// SIMATIC S7-200 project (STEP 7-Micro/WIN), CPU 224 CN REL 02.01

ORGANIZATION_BLOCK 补水控制:OB1
TITLE=我为200方给水净化工程设计了一个自动化控制系统，适用于自来水厂等场景。通过操作员按下启动按钮启动补水流程，并在未按下停止按钮时运行，确保供水质量和稳定性。
// 系统中涉及的物理设备包括补水泵1、补水泵2、进水阀、出水阀、余氯调节泵、水箱、启动按钮、停止按钮、水位传感器和阀门限位开关。
// Network 1开始，当启动按钮按下且停止按钮未按下时，若水位低传感器未触发，补水泵1启动，需通过定时器延时60个单位停止。
// Network 2中，补水泵2在水位高传感器未触发且标志位为真时启动，同样使用定时器延时停止。
// Network 3和Network 7通过定时器实现补水泵延时600个单位停止，确保水位恢复后泵不会立即停机。
// Network 16调用子程序，其中阀门控制根据阀门开限位和关限位控制进水阀和出水阀，要求动作在限位信号正确时执行。同时，进水阀和出水阀互锁防止同时开启。
// 当进水控制信号为真且阀门切换标志为假时，打开进水阀，以向水箱供水。
// 当出水控制信号为真时，打开出水阀，以排出水箱中的水。
// 余氯控制根据余氯浓度调节余氯调节泵，浓度低于7时启动，高于15时停止。
// 参数显示通过定时器每20个单位更新水质参数，并在触摸屏显示。
// PID控制根据补水泵状态调整模拟量输出，实现水流稳定。
// 
BEGIN
Network 1 // 网络标题
// 网络注释
LD     I0.0
AN     I0.1
AN     I0.2
AN     I2.1
AN     M0.0
LPS
A      T120
=      Q0.0
LPP
TON    T120, +60
Network 2
LD     I0.0
AN     I0.1
AN     I0.3
AN     I2.1
A      M0.0
LPS
A      T63
=      Q0.1
LPP
TON    T63, +60
Network 3
LD     Q0.0
AN     I0.2
AN     I0.3
AN     T37
AN     Q0.3
TON    T37, +600
Network 4
LD     SM0.0
MOVW   VW730, VW732
LDW<=  VW730, +0
O      M20.0
ALD
MOVW   +2880, VW730
Network 5
LD     T37
LD     Q0.1
CTU    C1, VW732
Network 6
LD     SM0.0
MOVW   C1, VW750
Network 7
LD     Q0.1
AN     I0.2
AN     I0.3
AN     Q0.2
AN     T38
TON    T38, +600
Network 8
LD     T38
LD     Q0.0
CTU    C2, VW732
Network 9
LD     SM0.0
MOVW   C2, VW754
Network 10
LD     C1
O      I0.2
O      M0.5
S      M0.0, 1
Network 11
LD     C2
O      I0.3
O      M0.6
R      M0.0, 1
Network 12
LD     I0.1
AN     I0.2
A      M0.4
O      M0.5
A      I0.0
=      Q0.2
Network 13
LD     I0.1
AN     I0.3
A      M0.4
A      I0.2
O      M0.6
A      I0.0
=      Q0.3
Network 14
LDW>   AIW2, +23480
R      M0.4, 1
Network 15
LDW<   AIW2, +14940
S      M0.4, 1
Network 16
LD     SM0.0
CALL   参数显示:SBR2
CALL   PID控制:SBR0
CALL   阀门控制:SBR1
CALL   余氯控制:SBR3
Network 17
LD     SM0.0
MOVW   VW1440, VW1446
-I     +3, VW1446
MOVW   VW1440, VW1500
+I     +0, VW1500
Network 18
LD     Q0.0
AN     Q0.3
AW>    VW1446, VW202
LPS
A      T45
S      M0.5, 1
LPP
TON    T45, +500
Network 19
LD     Q0.1
AN     Q0.2
AW>    VW1446, VW202
LPS
A      T46
S      M0.6, 1
LPP
TON    T46, +500
Network 20
LDW>=  VW202, VW1500
ON     I0.0
LPS
A      T48
R      M0.5, 2
LPP
TON    T48, +300
END_ORGANIZATION_BLOCK

SUBROUTINE_BLOCK PID控制:SBR0
TITLE=子程序注释
BEGIN
Network 1 // 网络标题
// 网络注释
LD     Q0.0
O      Q0.1
LPS
ITD    VW1440, AC1
LDW<=  VW1440, +0
O      M20.0
ALD
MOVW   +30, VW1440
LPP
DTR    AC1, VD1570
MOVR   VD1570, VD1572
*R     427.0, VD1572
MOVR   VD1572, VD504
/R     25600.0, VD504
Network 2
LDN    Q0.0
AN     Q0.1
MOVD   +0, VD504
Network 3
LD     SM0.0
MOVR   0.3, VD520
*R     1.0, VD520
Network 4
LD     SM0.0
MOVR   0.5, VD512
*R     1.0, VD512
Network 5
LD     SM0.0
MOVR   0.1, VD516
*R     1.0, VD516
Network 6
LD     SM0.0
XORD   AC0, AC0
MOVW   VW208, AC0
DTR    AC0, AC0
/R     25600.0, AC0
MOVR   AC0, VD500
Network 7
LD     SM0.0
PID    VB500, 0
Network 8
LD     SM0.0
MOVR   VD508, AC0
MOVR   VD508, AC0
*R     32000.0, AC0
TRUNC  AC0, AC0
MOVW   AC0, AQW0
END_SUBROUTINE_BLOCK

SUBROUTINE_BLOCK 阀门控制:SBR1
TITLE=
BEGIN
Network 1
LD     I0.4
AN     M0.3
=      Q0.4
A      I2.7
=      Q0.5
Network 2
LD     I0.4
A      M0.3
=      Q0.6
=      Q0.7
Network 3
LD     I1.0
AN     I1.2
AN     I0.7
AN     T39
TON    T39, +600
Network 4
LD     SM0.0
MOVW   VW718, VW720
LDW<=  VW718, +0
O      M20.0
ALD
MOVW   +7200, VW718
Network 5
LD     T39
LD     C4
CTU    C4, VW720
Network 6
LD     SM0.0
MOVW   C4, VW758
Network 7
LD     I1.3
A      I2.4
AN     I1.5
AN     I2.6
AN     T40
TON    T40, +600
Network 8
LD     SM0.0
MOVW   VW724, VW728
LDW<=  VW724, +0
O      M20.0
ALD
MOVW   +10, VW724
Network 9
LD     T40
LD     C5
CTU    C5, VW728
Network 10
LD     SM0.0
MOVW   C5, VW762
Network 11
LD     C4
S      M0.3, 1
Network 12
LD     C5
R      M0.3, 1
END_SUBROUTINE_BLOCK

SUBROUTINE_BLOCK 参数显示:SBR2
TITLE=
BEGIN
Network 1
LD     SM0.0
AN     M1.4
TON    T50, +20
Network 2
LD     T50
EU
=      M1.4
Network 3
LD     M1.4
+R     1.0, VD2000
Network 4
LDR=   VD2000, 4.0
MOVR   0.0, VD2000
Network 5
LDR=   VD2000, 1.0
MOVW   AIW0, VW160
MOVW   AIW2, VW220
MOVW   AIW4, VW420
MOVW   AIW6, VW620
Network 6
LDR=   VD2000, 2.0
MOVW   AIW0, VW164
MOVW   AIW2, VW230
MOVW   AIW4, VW430
MOVW   AIW6, VW630
Network 7
LDR=   VD2000, 3.0
MOVW   AIW0, VW170
MOVW   AIW2, VW240
MOVW   AIW4, VW440
MOVW   AIW6, VW640
Network 8
LD     M1.4
MOVW   VW160, VW162
/I     +3, VW162
MOVW   VW164, VW166
/I     +3, VW166
MOVW   VW170, VW172
/I     +3, VW172
MOVW   VW162, VW180
+I     VW166, VW180
MOVW   VW180, VW194
+I     VW172, VW194
Network 9
LD     M1.4
MOVW   VW220, VW222
/I     +3, VW222
MOVW   VW230, VW232
/I     +3, VW232
MOVW   VW240, VW242
/I     +3, VW242
MOVW   VW222, VW250
+I     VW232, VW250
MOVW   VW250, VW204
+I     VW242, VW204
Network 10
LD     M1.4
MOVW   VW420, VW422
/I     +3, VW422
MOVW   VW430, VW432
/I     +3, VW432
MOVW   VW440, VW442
/I     +3, VW442
MOVW   VW422, VW450
+I     VW432, VW450
MOVW   VW450, VW404
+I     VW442, VW404
Network 11
LD     M1.4
MOVW   VW620, VW622
/I     +3, VW622
MOVW   VW630, VW632
/I     +3, VW632
MOVW   VW640, VW642
/I     +3, VW642
MOVW   VW622, VW650
+I     VW632, VW650
MOVW   VW650, VW604
+I     VW642, VW604
Network 12
LD     SM0.0
AN     M1.5
TON    T51, +20
Network 13
LD     T51
EU
=      M1.5
Network 14
LD     SM0.0
LPS
AW<=   VW194, +6400
MOVW   +0, VW198
LRD
AW<=   VW204, +6400
MOVW   +0, VW208
LRD
AW<=   VW404, +6400
MOVW   +0, VW408
LPP
AW<=   VW604, +6400
MOVW   +0, VW608
Network 15
LD     M1.5
LPS
AW>=   VW194, +6400
MOVW   VW194, VW198
-I     +6400, VW198
LRD
AW>=   VW204, +6400
MOVW   VW204, VW208
-I     +6400, VW208
LRD
AW>=   VW404, +6400
MOVW   VW404, VW408
-I     +6400, VW408
LPP
AW>=   VW604, +6400
MOVW   VW604, VW608
-I     +6400, VW608
Network 16
LD     SM0.0
AN     M1.6
TON    T52, +20
Network 17
LD     T52
EU
=      M1.6
Network 18
LD     M1.6
LPS
AW<=   VW194, +6400
LPS
NOT
AW>=   VW194, +32000
LPS
NOT
MOVW   VW198, VW192
DIV    +13, VD190
LPP
MOVW   +2000, VW192
LPP
MOVW   +0, VW192
LRD
AW<=   VW204, +6400
LPS
NOT
AW>=   VW204, +32000
LPS
NOT
MOVW   VW208, VW202
DIV    +427, VD200
LPP
MOVW   +60, VW202
LPP
MOVW   +0, VW202
LRD
AW<=   VW404, +6400
LPS
NOT
AW>=   VW404, +32000
LPS
NOT
MOVW   VW408, VW402
DIV    +160, VD400
LPP
MOVW   +160, VW402
LPP
MOVW   +0, VW402
LPP
AW<=   VW604, +6400
LPS
NOT
AW>=   VW604, +32000
LPS
NOT
MOVW   VW608, VW602
DIV    +160, VD600
LPP
MOVW   +160, VW602
LPP
MOVW   +0, VW602
END_SUBROUTINE_BLOCK

SUBROUTINE_BLOCK 余氯控制:SBR3
TITLE=
BEGIN
Network 1
LDW>   VW192, +15
R      M0.7, 1
Network 2
LD     Q1.0
A      SM0.4
LD     C16
OW>    VW192, +15
CTU    C16, +20
Network 3
LD     M0.7
=      Q1.0
Network 4
LD     C16
R      M0.7, 1
Network 5
LD     C18
S      M0.7, 1
Network 6
LDN    Q1.0
A      SM0.4
AW<    VW192, +7
LD     Q1.0
CTU    C18, +60
END_SUBROUTINE_BLOCK
